PROGRAM Axis02_X_1
VAR
	Axis02: AXIS_REF;											//회전축
	Axis02_MC_Home: FB_HomeBeforeMoveAX8000:=(channel:=2);
	Axis02_MC_Power: MC_Power;
	Axis02_Status: MC_ReadStatus;
	Axis02_Position_Read: MC_ReadActualPosition;
	Axis02_Velocity_Read: MC_ReadActualVelocity;
	Axis02_Reset: MC_Reset;										//모터 알람 리셋
	Axis02_Stop: MC_Stop;										//모터 정지
	Axis02_Press_Move: MC_MoveAbsolute;
	Axis02_Home_Pos_Move: MC_MoveAbsolute;
	Axis02_Wait_Pos_Move: MC_MoveAbsolute;
	Axis02_Target_Pos_Move: MC_MoveAbsolute;
	Axis02_Work_End_Move: MC_MoveAbsolute;
	Axis02_Jog: MC_Jog;
	
	Always_ON				:	BOOL	:=TRUE	;//상시 ON
	Always_OFF				:	BOOL	:=FALSE	;//상시 OFF
	Home_Interlock			:	Bool	;
	Home_Pos_Interlock		: 	BOOL	;
	Wait_Pos_Interlock		:	BOOL	;
	Target_Pos_Interlock	:	BOOL	;
	Work_End_POs_Interlock	:	BOOL	;
	
	Axis02_Calibration: MC_MoveAbsolute;
	Calibration_Pos_Interlock: BOOL;
	Axis02_Tool_Change: MC_MoveAbsolute;
	Axis02_Target_Move02: MC_MoveSuperImposed;
	Axis02_Target_Pos_Move02: MC_GearInVelo;
	Axis02_Move: MC_GearInVelo;
	test: BOOL;

	MC_GearIn_0: MC_GearIn;
	test01: BOOL;
	MC_MoveVelocity_0: MC_MoveVelocity;
	test02: BOOL;
END_VAR
VAR // added by the converter: edge detectors and wires of the graphical bodies
    _rt1, _rt2, _rt3, _rt4, _rt5, _rt6, _rt7 : R_TRIG;
END_VAR

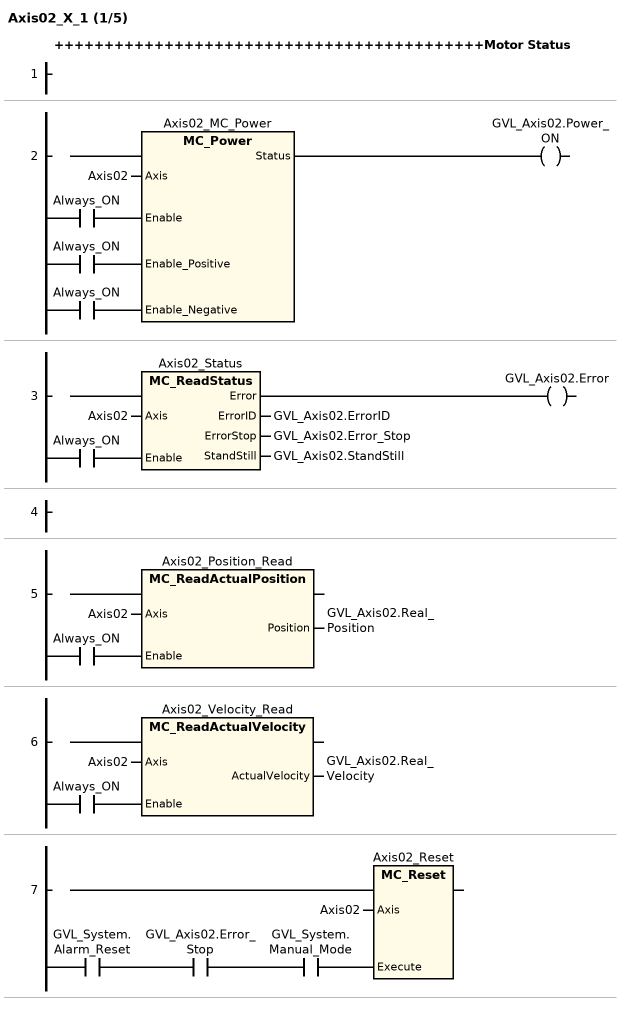
// NETWORK 1: +++++++++++++++++++++++++++++++++++++++++++Motor Status

// NETWORK 2
Axis02_MC_Power(
    Axis := Axis02,
    Enable := Always_ON,
    Enable_Positive := Always_ON,
    Enable_Negative := Always_ON); // MC_Power
GVL_Axis02.Power_ON := Axis02_MC_Power.Status;

// NETWORK 3
Axis02_Status(
    Axis := Axis02,
    Enable := Always_ON,
    Error => GVL_Axis02.Error,
    ErrorID => GVL_Axis02.ErrorID,
    ErrorStop => GVL_Axis02.Error_Stop,
    StandStill => GVL_Axis02.StandStill); // MC_ReadStatus

// NETWORK 4

// NETWORK 5
Axis02_Position_Read(Axis := Axis02, Enable := Always_ON, Position => GVL_Axis02.Real_Position); // MC_ReadActualPosition

// NETWORK 6
Axis02_Velocity_Read(Axis := Axis02, Enable := Always_ON, ActualVelocity => GVL_Axis02.Real_Velocity); // MC_ReadActualVelocity

// NETWORK 7
Axis02_Reset(Axis := Axis02, Execute := GVL_System.Alarm_Reset AND GVL_Axis02.Error_Stop AND GVL_System.Manual_Mode); // MC_Reset

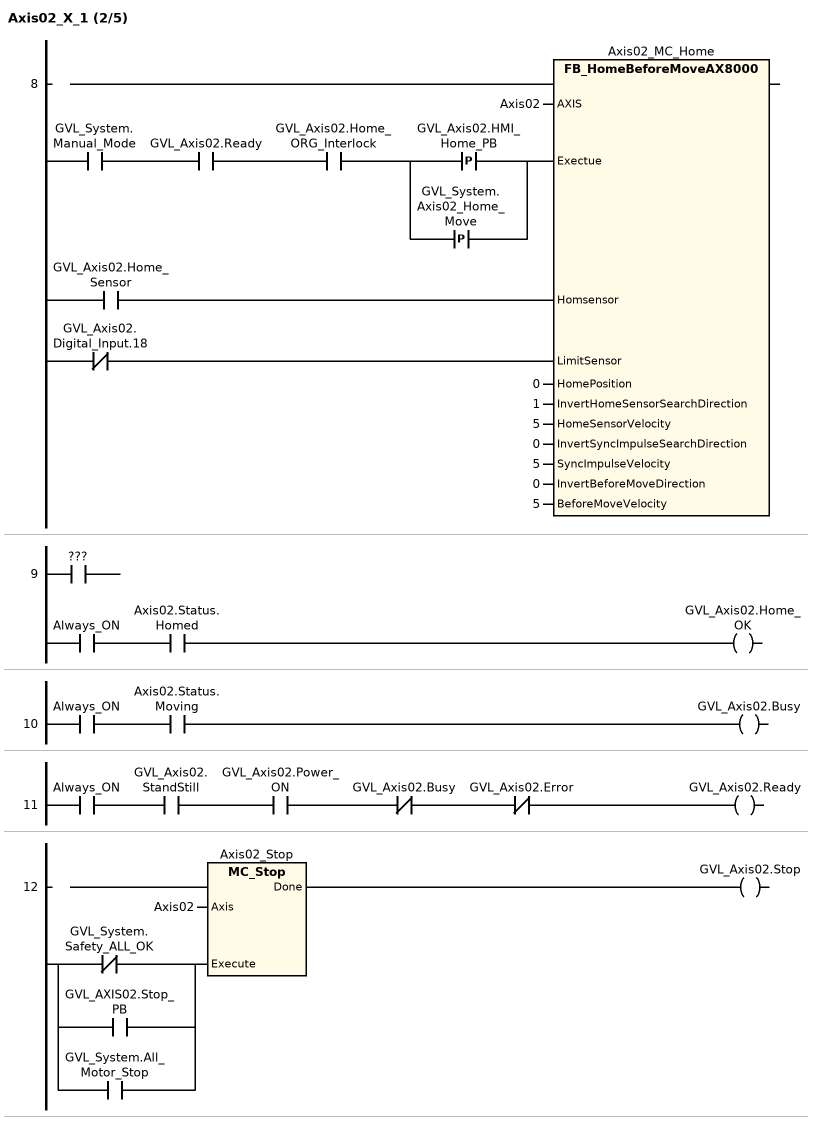
// NETWORK 8
_rt1(CLK := GVL_Axis02.HMI_Home_PB);
_rt2(CLK := GVL_System.Axis02_Home_Move);
Axis02_MC_Home(
    AXIS := Axis02,
    Exectue := GVL_System.Manual_Mode AND GVL_Axis02.Ready AND GVL_Axis02.Home_ORG_Interlock AND (_rt1.Q OR _rt2.Q),
    Homsensor := GVL_Axis02.Home_Sensor,
    LimitSensor := NOT GVL_Axis02.Digital_Input.18,
    HomePosition := 0,
    InvertHomeSensorSearchDirection := 1,
    HomeSensorVelocity := 5,
    InvertSyncImpulseSearchDirection := 0,
    SyncImpulseVelocity := 5,
    InvertBeforeMoveDirection := 0,
    BeforeMoveVelocity := 5); // FB_HomeBeforeMoveAX8000

// NETWORK 9
GVL_Axis02.Home_OK := Always_ON AND Axis02.Status.Homed;

// NETWORK 10
GVL_Axis02.Busy := Always_ON AND Axis02.Status.Moving;

// NETWORK 11
GVL_Axis02.Ready := Always_ON AND GVL_Axis02.StandStill AND GVL_Axis02.Power_ON AND NOT GVL_Axis02.Busy AND NOT GVL_Axis02.Error;

// NETWORK 12
Axis02_Stop(Axis := Axis02, Execute := NOT GVL_System.Safety_ALL_OK OR GVL_AXIS02.Stop_PB OR GVL_System.All_Motor_Stop); // MC_Stop
GVL_Axis02.Stop := Axis02_Stop.Done;

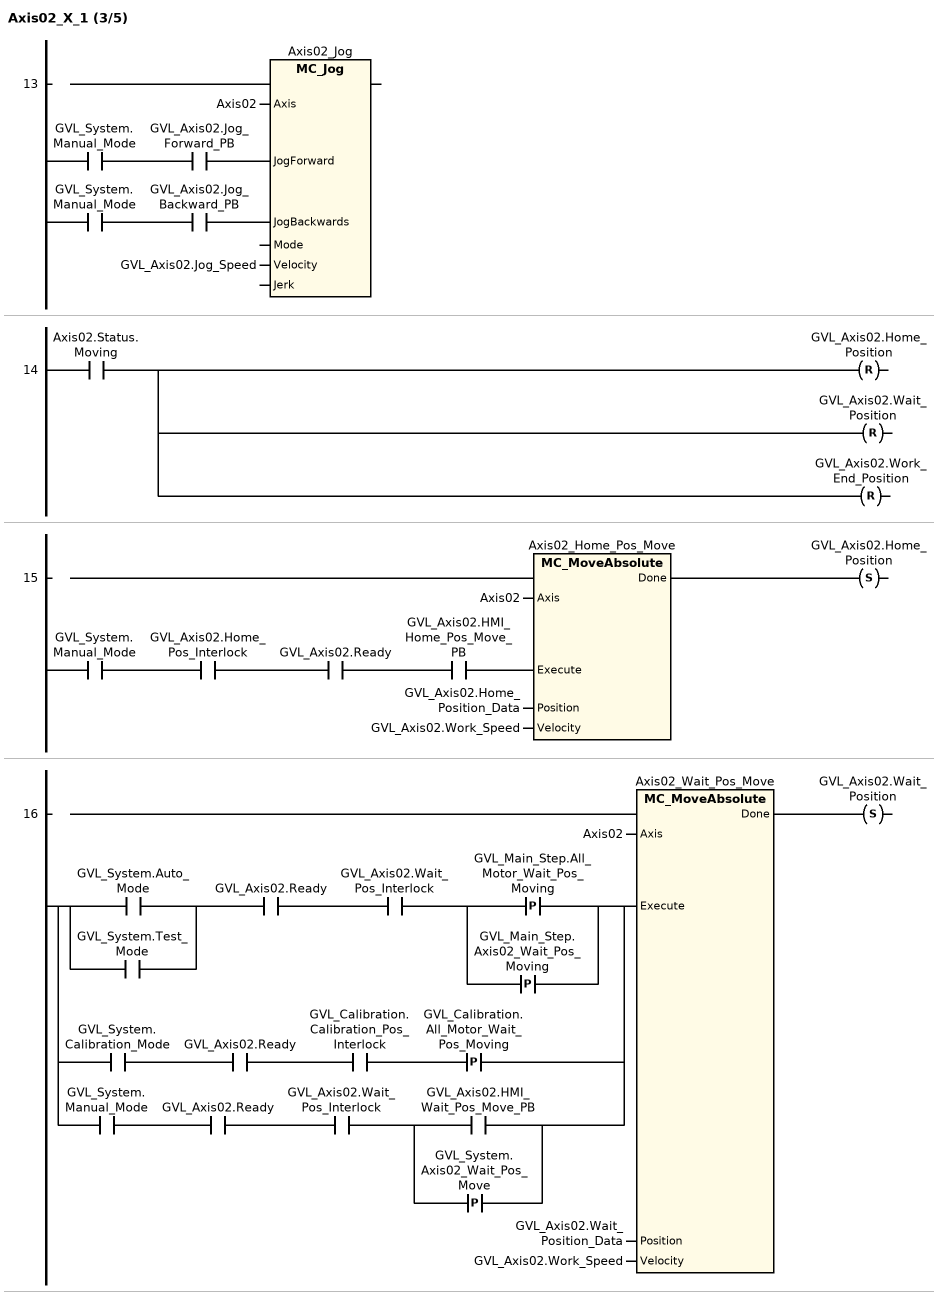
// NETWORK 13
Axis02_Jog(
    Axis := Axis02,
    JogForward := GVL_System.Manual_Mode AND GVL_Axis02.Jog_Forward_PB,
    JogBackwards := GVL_System.Manual_Mode AND GVL_Axis02.Jog_Backward_PB,
    Velocity := GVL_Axis02.Jog_Speed); // MC_Jog

// NETWORK 14
GVL_Axis02.Home_Position R= Axis02.Status.Moving;
GVL_Axis02.Wait_Position R= Axis02.Status.Moving;
GVL_Axis02.Work_End_Position R= Axis02.Status.Moving;

// NETWORK 15
Axis02_Home_Pos_Move(
    Axis := Axis02,
    Execute := GVL_System.Manual_Mode AND GVL_Axis02.Home_Pos_Interlock AND GVL_Axis02.Ready AND GVL_Axis02.HMI_Home_Pos_Move_PB,
    Position := GVL_Axis02.Home_Position_Data,
    Velocity := GVL_Axis02.Work_Speed); // MC_MoveAbsolute
GVL_Axis02.Home_Position S= Axis02_Home_Pos_Move.Done;

// NETWORK 16
_rt3(CLK := GVL_Main_Step.All_Motor_Wait_Pos_Moving);
_rt4(CLK := GVL_Main_Step.Axis02_Wait_Pos_Moving);
_rt5(CLK := GVL_Calibration.All_Motor_Wait_Pos_Moving);
_rt6(CLK := GVL_System.Axis02_Wait_Pos_Move);
Axis02_Wait_Pos_Move(
    Axis := Axis02,
    Execute := (GVL_System.Auto_Mode OR GVL_System.Test_Mode) AND GVL_Axis02.Ready AND GVL_Axis02.Wait_Pos_Interlock AND (_rt3.Q OR _rt4.Q) OR GVL_System.Calibration_Mode AND GVL_Axis02.Ready AND GVL_Calibration.Calibration_Pos_Interlock AND _rt5.Q OR GVL_System.Manual_Mode AND GVL_Axis02.Ready AND GVL_Axis02.Wait_Pos_Interlock AND (GVL_Axis02.HMI_Wait_Pos_Move_PB OR _rt6.Q),
    Position := GVL_Axis02.Wait_Position_Data,
    Velocity := GVL_Axis02.Work_Speed); // MC_MoveAbsolute
GVL_Axis02.Wait_Position S= Axis02_Wait_Pos_Move.Done;

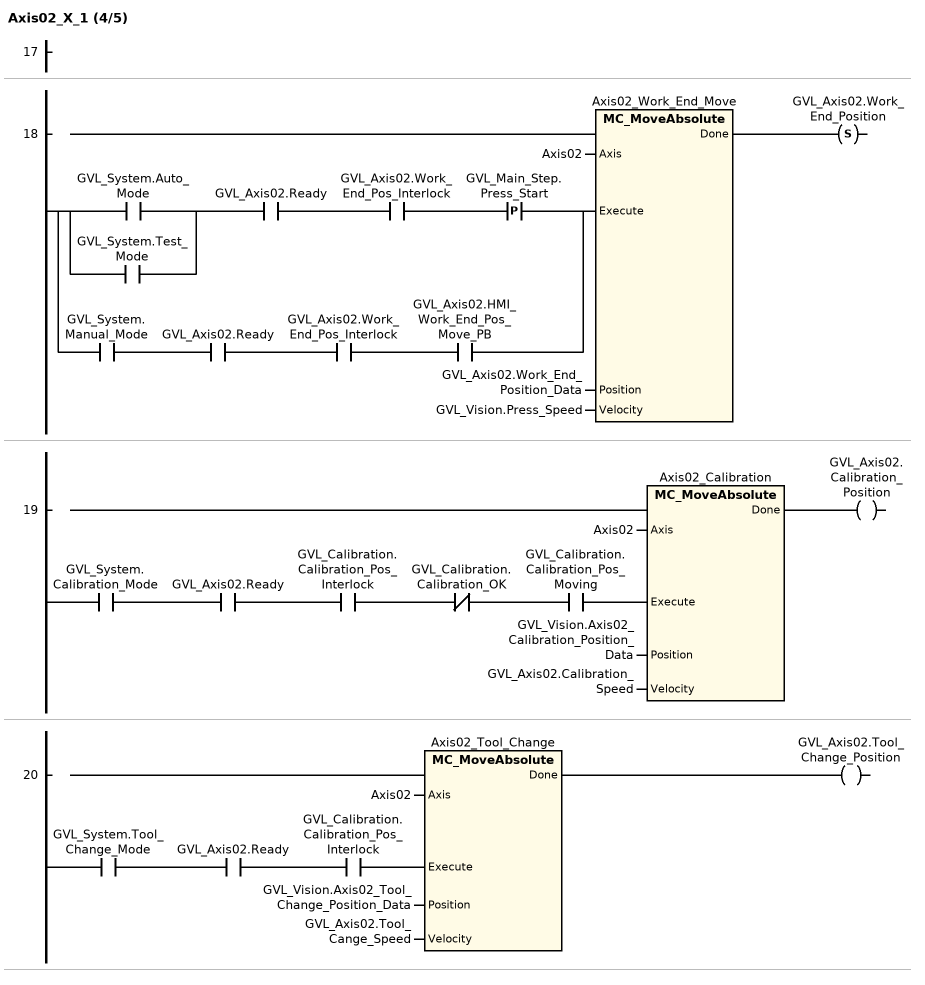
// NETWORK 17

// NETWORK 18
_rt7(CLK := GVL_Main_Step.Press_Start);
Axis02_Work_End_Move(
    Axis := Axis02,
    Execute := (GVL_System.Auto_Mode OR GVL_System.Test_Mode) AND GVL_Axis02.Ready AND GVL_Axis02.Work_End_Pos_Interlock AND _rt7.Q OR GVL_System.Manual_Mode AND GVL_Axis02.Ready AND GVL_Axis02.Work_End_Pos_Interlock AND GVL_Axis02.HMI_Work_End_Pos_Move_PB,
    Position := GVL_Axis02.Work_End_Position_Data,
    Velocity := GVL_Vision.Press_Speed); // MC_MoveAbsolute
GVL_Axis02.Work_End_Position S= Axis02_Work_End_Move.Done;

// NETWORK 19
Axis02_Calibration(
    Axis := Axis02,
    Execute := GVL_System.Calibration_Mode AND GVL_Axis02.Ready AND GVL_Calibration.Calibration_Pos_Interlock AND NOT GVL_Calibration.Calibration_OK AND GVL_Calibration.Calibration_Pos_Moving,
    Position := GVL_Vision.Axis02_Calibration_Position_Data,
    Velocity := GVL_Axis02.Calibration_Speed); // MC_MoveAbsolute
GVL_Axis02.Calibration_Position := Axis02_Calibration.Done;

// NETWORK 20
Axis02_Tool_Change(
    Axis := Axis02,
    Execute := GVL_System.Tool_Change_Mode AND GVL_Axis02.Ready AND GVL_Calibration.Calibration_Pos_Interlock,
    Position := GVL_Vision.Axis02_Tool_Change_Position_Data,
    Velocity := GVL_Axis02.Tool_Cange_Speed); // MC_MoveAbsolute
GVL_Axis02.Tool_Change_Position := Axis02_Tool_Change.Done;

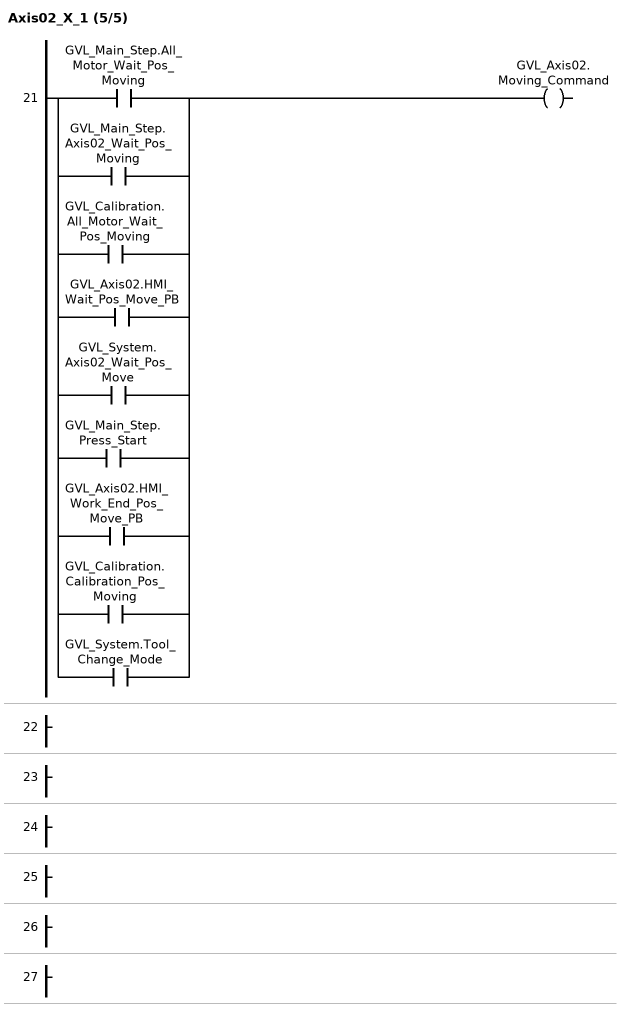
// NETWORK 21
GVL_Axis02.Moving_Command := GVL_Main_Step.All_Motor_Wait_Pos_Moving OR GVL_Main_Step.Axis02_Wait_Pos_Moving OR GVL_Calibration.All_Motor_Wait_Pos_Moving OR GVL_Axis02.HMI_Wait_Pos_Move_PB OR GVL_System.Axis02_Wait_Pos_Move OR GVL_Main_Step.Press_Start OR GVL_Axis02.HMI_Work_End_Pos_Move_PB OR GVL_Calibration.Calibration_Pos_Moving OR GVL_System.Tool_Change_Mode;

// NETWORK 22

// NETWORK 23

// NETWORK 24

// NETWORK 25

// NETWORK 26

// NETWORK 27

END_PROGRAM

(* stored: Version 1.1.0.1, ProductVersion 3.1.4024.15
   POU Axis02_X_1: Id {5dee82d8-93f1-467b-b199-b926e0393542}, SpecialFunc None *)
